Universal Robots PolyScope program: taskboard_belt_v7.urp

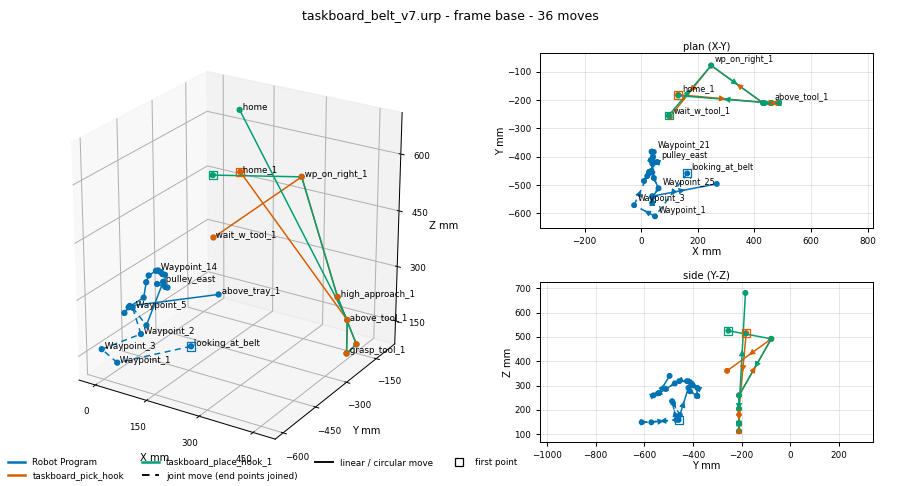
[picture p0: tool path of taskboard_belt_v7.urp in frame base, 36 of 39 moves have a stored position in this frame; points joined in program order, loops and branches not executed]
Program taskboard_belt_v7 (installation=default directory=/programs/wrs2020 createdIn=3.8.0.61336 lastSavedIn=5.10.0.106288 robotSerialNumber=20205500607)
Calibrated DH parameters: a=[0.000096, -0.337, -0.383372, 0.000118, 0.000015, 0]; d=[0.162724, 79.377998, -95.545185, 16.300583, 0.099689, 0.099499]; alpha=[1.569249, 0.003272, 0.005201, 1.570041, -1.570219, 0]; deltaTheta=[0, 0.65664, 5.410619, 0.215927, -0.000001, 0]
Robot Program (runOnlyOnce=true)
  SuppressedNode
    Call taskboard_pick_hook
  MoveJ speed 60 deg/s, acceleration 80 deg/s^2 (useActiveTCP=false) tcp=gripper_85_tip; feature=Base
    currentpose := get_actual_joint_positions()
    Waypoint Waypoint (Variable): variable=currentpose
    Waypoint looking_at_belt: TCP in base x=162.548 y=-458.764 z=158.73 mm, rx=-1.6745 ry=-2.0805 rz=0.6897 rad; joints [112.15, -80.245, 110.523, -113.873, -125.384, 101.857] deg; TCP offset x=0 y=0 z=165 mm, rx=0 ry=0 rz=0 rad
  Popup Message (haltProgram=false message=start sequence with a_bot (simultaneous start) inputType=Text)
  SuppressedNode
    MoveJ speed 150 deg/s, acceleration 120 deg/s^2 (useActiveTCP=false) tcp=TCP; feature=Base
      Waypoint Waypoint_6: TCP in base x=127.08 y=-413.334 z=291.81 mm, rx=-0.7232 ry=-2.7798 rz=0.8385 rad; joints [93.391, -90.83, 132.55, -160.801, -107.268, 28.161] deg
      Waypoint Waypoint_7: TCP in base x=29.418 y=-413.334 z=291.81 mm, rx=-1.1848 ry=-2.5289 rz=0.748 rad; joints [80.663, -93.425, 133.978, -156.473, -111.093, 36.06] deg
  Wait Sleep waitTime=1.5
  MoveJ speed 180 deg/s, acceleration 120 deg/s^2 (useActiveTCP=false) tcp=gripper_85_tip; feature=Base
    Waypoint Waypoint_1: motionParameters(blendRadius=0.01); TCP in base x=48.773 y=-610.591 z=148.889 mm, rx=-1.4737 ry=-2.1715 rz=0.79 rad; joints [97.835, -68.658, 103.848, -135.751, -128.895, 72.525] deg; TCP offset x=0 y=0 z=165 mm, rx=0 ry=0 rz=0 rad
    Waypoint Waypoint_3: motionParameters(blendRadius=0.015); TCP in base x=-25.071 y=-571.131 z=148.885 mm, rx=-1.7354 ry=-1.8972 rz=0.6872 rad; joints [91.414, -71.26, 105.056, -125.967, -130.041, 85.588] deg
    Waypoint Waypoint_2: motionParameters(blendRadius=0.01); TCP in base x=21.111 y=-468.4 z=159.302 mm, rx=-2.0556 ry=-1.7797 rz=0.5274 rad; joints [92.758, -84.336, 113.518, -115.329, -119.963, 102.011] deg
    Waypoint Waypoint_5: motionParameters(blendRadius=0.01); TCP in base x=9.828 y=-485.674 z=235.678 mm, rx=-2.1579 ry=-1.6243 rz=0.4873 rad; joints [91.069, -84.715, 100.871, -98.824, -119.366, 108.969] deg
    Waypoint Waypoint_4: TCP in base x=27.871 y=-453.713 z=178.666 mm, rx=-1.9239 ry=-1.8837 rz=0.5527 rad; joints [94.601, -87.608, 114.765, -114.053, -121.77, 96.675] deg
  MoveL speed 1000 mm/s, acceleration 600 mm/s^2 (useActiveTCP=false) tcp=TCP; feature=Base
    Waypoint pulley_east: motionParameters(blendRadius=0.026); TCP in base x=55.998 y=-418.531 z=290.523 mm, rx=-1.8278 ry=-1.8742 rz=0.615 rad; joints [87.749, -91.494, 125.705, -126.247, -126.512, 85.659] deg
    Waypoint pulley_seast: motionParameters(blendRadius=0.001); TCP in base x=33.502 y=-412.204 z=276.546 mm, rx=-1.9192 ry=-1.9671 rz=0.4925 rad; joints [82.773, -92.565, 128.49, -130.133, -117.87, 80.345] deg
    Waypoint Waypoint_21: motionParameters(blendRadius=0.001); TCP in base x=44.298 y=-382.864 z=257.805 mm, rx=-1.6371 ry=-2.0929 rz=0.685 rad; joints [85.273, -92.843, 136.557, -146.414, -124.378, 67.476] deg
    Waypoint Waypoint_18: motionParameters(blendRadius=0.006); TCP in base x=37.055 y=-382.126 z=257.637 mm, rx=-1.629 ry=-2.1021 rz=0.687 rad; joints [84.068, -92.976, 137.087, -147.929, -123.937, 65.465] deg
    Waypoint Waypoint_17: motionParameters(blendRadius=0.005); TCP in base x=37.055 y=-382.126 z=290.533 mm, rx=-1.629 ry=-2.1021 rz=0.687 rad; joints [84.087, -97.119, 134.374, -141.084, -123.927, 65.444] deg
    Waypoint Waypoint_16: motionParameters(blendRadius=0.005); TCP in base x=41.622 y=-399.96 z=300.439 mm, rx=-1.7118 ry=-2.0151 rz=0.6578 rad; joints [85.295, -95.468, 129.851, -133.893, -125.21, 72.993] deg
    Waypoint Waypoint_15: motionParameters(blendRadius=0.002); TCP in base x=40.113 y=-404.528 z=307.021 mm, rx=-1.7118 ry=-2.0151 rz=0.6578 rad; joints [85.13, -95.461, 128.724, -132.891, -125.179, 72.788] deg
    Waypoint Waypoint_14: motionParameters(blendRadius=0.003); TCP in base x=37.055 y=-412.061 z=313.946 mm, rx=-1.7118 ry=-2.0151 rz=0.6578 rad; joints [84.782, -95.052, 127.233, -132.056, -125.116, 72.363] deg
    Waypoint Waypoint_13: motionParameters(blendRadius=0.003); TCP in base x=39.115 y=-424.305 z=318.144 mm, rx=-1.7118 ry=-2.0151 rz=0.6578 rad; joints [85.23, -93.633, 125.136, -131.064, -125.187, 72.904] deg
    Waypoint Waypoint_12: motionParameters(blendRadius=0.003); TCP in base x=39.115 y=-456.158 z=318.144 mm, rx=-1.7118 ry=-2.0151 rz=0.6578 rad; joints [85.574, -89.225, 120.79, -130.878, -125.234, 73.332] deg
    Waypoint after_pulley: motionParameters(blendRadius=0.005); TCP in base x=44.33 y=-474.815 z=308.597 mm, rx=-1.7118 ry=-2.0151 rz=0.6578 rad; joints [86.4, -85.893, 118.745, -131.572, -125.36, 74.349] deg
    Waypoint Waypoint_25: motionParameters(blendRadius=0.01); TCP in base x=61.142 y=-511.386 z=285.958 mm, rx=-1.7746 ry=-1.9444 rz=0.6341 rad; joints [88.659, -79.129, 113.407, -128.412, -126.069, 82.135] deg
    Waypoint Waypoint_26: motionParameters(blendRadius=0.005); TCP in base x=38.979 y=-543.773 z=267.745 mm, rx=-1.7746 ry=-1.9444 rz=0.6341 rad; joints [86.354, -74.004, 110.475, -132.267, -125.862, 79.326] deg
    Waypoint Waypoint_27: TCP in base x=38.979 y=-562.173 z=259.861 mm, rx=-1.7746 ry=-1.9444 rz=0.6341 rad; joints [86.471, -71.214, 107.961, -132.453, -125.87, 79.482] deg
    Waypoint Waypoint_28: motionParameters(blendRadius=0.005); TCP in base x=38.979 y=-539.175 z=269.332 mm, rx=-1.7746 ry=-1.9444 rz=0.6341 rad; joints [86.323, -74.676, 111.111, -132.256, -125.86, 79.286] deg
    Waypoint above_tray_1: motionParameters(blendRadius=0.03); TCP in base x=266.866 y=-496.012 z=339.711 mm, rx=-1.7965 ry=-1.8026 rz=0.6723 rad; joints [111.069, -74.141, 92.89, -90.937, -127.591, 116.905] deg
    SuppressedNode
      Waypoint drop_belt: motionParameters(blendRadius=0.005); TCP in base x=230.499 y=-434.048 z=320.965 mm, rx=1.7763 ry=1.8835 rz=-0.8946 rad; joints [106.189, -83.529, 124.565, -171.821, -108.616, 96.025] deg
    SuppressedNode
      Waypoint above_tray_1: motionParameters(blendRadius=0.009); TCP in base x=266.866 y=-496.012 z=339.711 mm, rx=-1.7965 ry=-1.8026 rz=0.6723 rad; joints [111.069, -74.141, 92.89, -90.937, -127.591, 116.905] deg
    SuppressedNode
      Waypoint look_at_result: TCP in base x=266.865 y=-496.017 z=308.801 mm, rx=-1.7965 ry=-1.8026 rz=0.6723 rad; joints [111.063, -72.645, 95.725, -95.254, -127.586, 116.932] deg
  SuppressedNode
    Call taskboard_place_hook_1
SubProgram -> taskboard_pick_hook
SubProgram -> taskboard_place_hook_1
SubProgram taskboard_pick_hook (keepSynchronizedWithDisk=false) programFile=/programs/wrs2020/taskboard_pick_hook.urp
  URCap Gripper (Robotiq_Grippers, Robotiq Inc.) dataModel(position=0.0, force=100.0, speed=100.0, positionInDouble=0.0, forceInDouble=100.0, speedInDouble=100.0, slaveIds=[9], blocking=false)
  MoveJ speed 60 deg/s, acceleration 80 deg/s^2 (useActiveTCP=true) feature=Base
    currentpose := get_actual_joint_positions()
    Waypoint Waypoint (Variable): variable=currentpose
  MoveL speed 800 mm/s, acceleration 800 mm/s^2 (useActiveTCP=false) tcp=TCP; feature=Base
    Waypoint home_1: TCP in base x=130.649 y=-180.735 z=515.945 mm, rx=-0.0119 ry=-3.1403 rz=-0.0318 rad; joints [89.95, -120.316, 80.212, -48.703, -89.953, 0.003] deg; TCP offset x=0 y=0 z=165 mm, rx=0 ry=0 rz=0 rad
    Waypoint above_tool_1: TCP in base x=459.162 y=-210.304 z=204.201 mm, rx=1.7463 ry=-1.7306 rz=-0.729 rad; joints [145.218, -68.652, 102.912, -84.042, -115.104, -26.034] deg
    Waypoint grasp_tool_1: TCP in base x=459.162 y=-210.304 z=112.252 mm, rx=1.7463 ry=-1.7306 rz=-0.729 rad; joints [145.194, -60.295, 107.111, -96.572, -115.081, -25.972] deg
    URCap Gripper (Robotiq_Grippers, Robotiq Inc.) dataModel(position=100.0, force=100.0, speed=100.0, positionInDouble=100.0, forceInDouble=100.0, speedInDouble=100.0, slaveIds=[9], blocking=true)
  MoveL speed 800 mm/s, acceleration 800 mm/s^2 (useActiveTCP=false) tcp=TCP; feature=Base
    Waypoint before_tool_1: TCP in base x=486.311 y=-210.304 z=144.711 mm, rx=1.7463 ry=-1.7306 rz=-0.729 rad; joints [146.732, -60.807, 101.299, -89.72, -114.09, -24.722] deg
    Waypoint high_approach_1: motionParameters(blendRadius=0.05); TCP in base x=430.518 y=-210.304 z=259.484 mm, rx=2.0705 ry=-2.0633 rz=-0.2652 rad; joints [140.289, -82.581, 114.687, -110.586, -100.48, -38.868] deg
    Waypoint wp_on_right_1: motionParameters(blendRadius=0.05); TCP in base x=247.136 y=-77.743 z=492.156 mm, rx=-1.0893 ry=2.9411 rz=0.0437 rad; joints [131.739, -127.117, 113.467, -74.929, -88.981, 0.805] deg
    Waypoint wait_w_tool_1: TCP in base x=101.033 y=-259.473 z=360.486 mm, rx=0.2423 ry=3.1043 rz=-0.0456 rad; joints [81.332, -124.8, 108.438, -75.156, -88.116, -0.001] deg; TCP offset x=0 y=0 z=165 mm, rx=0 ry=0 rz=0 rad
SubProgram taskboard_place_hook_1 (keepSynchronizedWithDisk=false) programFile=/programs/wrs2020/taskboard_place_hook.urp
  MoveJ speed 60 deg/s, acceleration 80 deg/s^2 (useActiveTCP=true) feature=Base
    currentpose := get_actual_joint_positions()
    Waypoint Waypoint (Variable): variable=currentpose
  MoveL speed 800 mm/s, acceleration 800 mm/s^2 (useActiveTCP=false) tcp=TCP; feature=Base
    Waypoint wait_w_tool: TCP in base x=96.884 y=-254.304 z=525.339 mm, rx=0.2424 ry=3.1043 rz=-0.0456 rad; joints [81.331, -124.8, 108.44, -75.158, -88.117, 0] deg; TCP offset x=0 y=0 z=0 mm, rx=0 ry=0 rz=0 rad
    Waypoint Waypoint_right: motionParameters(blendRadius=0.05); TCP in base x=247.136 y=-77.743 z=492.156 mm, rx=-1.0893 ry=2.9411 rz=0.0437 rad; joints [131.739, -127.117, 113.467, -74.929, -88.981, 0.805] deg
    Waypoint high_approach: motionParameters(blendRadius=0.05); TCP in base x=430.518 y=-210.304 z=259.484 mm, rx=2.0705 ry=-2.0633 rz=-0.2652 rad; joints [140.289, -82.581, 114.687, -110.586, -100.48, -38.868] deg
    Waypoint before_tool: motionParameters(blendRadius=0.005); TCP in base x=486.311 y=-210.304 z=144.711 mm, rx=1.7463 ry=-1.7306 rz=-0.729 rad; joints [146.732, -60.807, 101.299, -89.72, -114.09, -24.722] deg
    Waypoint grasp_tool: TCP in base x=459.162 y=-210.304 z=112.252 mm, rx=1.7463 ry=-1.7306 rz=-0.729 rad; joints [145.194, -60.295, 107.111, -96.572, -115.081, -25.972] deg
    URCap Gripper (Robotiq_Grippers, Robotiq Inc.) dataModel(position=0.0, force=100.0, speed=100.0, positionInDouble=0.0, forceInDouble=100.0, speedInDouble=100.0, slaveIds=[9], blocking=true)
    Waypoint above_tool: TCP in base x=459.162 y=-210.304 z=204.201 mm, rx=1.7463 ry=-1.7306 rz=-0.729 rad; joints [145.218, -68.652, 102.912, -84.042, -115.104, -26.034] deg
    Waypoint home: TCP in base x=130.839 y=-184.016 z=680.9 mm, rx=-0.0118 ry=-3.1403 rz=-0.0318 rad; joints [89.955, -120.323, 80.216, -48.702, -89.952, 0.003] deg
